FUNCTION_BLOCK SR (* IEC 61131-3 Table 34,#1 *)
  (* Standard: 61131-3 *)
  (* Version 0.0, 2004-12-15, JHC, Rockwell Automation, Converted from SRC format. *)
  (* Compiler header: package fb.rt.plc; *)
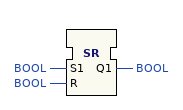
  VAR_INPUT
    S1 : BOOL;
    R : BOOL;
  END_VAR
  VAR_OUTPUT
    Q1 : BOOL;
  END_VAR
  ALGORITHM REQ IN ST:
IF S1 THEN Q1:=true;
ELSIF R THEN Q1:=false;
END_IF;
  END_ALGORITHM
END_FUNCTION_BLOCK
